Staubli VAL3: francais.pjx

--- francais.pjx ---
Parameters version=s7.1 stackSize=5000 millimeterUnit=true
Program file=message.pgx
Program file=page.pgx
Data file=francais.dtx

--- message.pgx ---
public program message(string& message[], num index)
// English IF message
begin
  // lenght of message
  //
  switch index
    case 0
      message="Voulez-vous entrer dans le:"
    break
    case 1
      message="< SI ASSISTANT >"
    break
    case 2
      message="Sélect. le type de condition pour vérifier"
    break
    case 3
      message="Sélect. l'Entrée"
    break
    case 4
      message="Sélect. la Sortie"
    break
    case 5
      message="Sélect. L'entrée EMAP"
    break
    case 6
      message="Sélect. la voie comment faire fonctionner l'instruction"
    break
    case 7
      message="Sélect. l'instruction pour associer vers le:"
    break
    case 8
      message="Sélect. de la liste le: "
    break
  endSwitch
end

--- page.pgx ---
public program page(string& menuname[], num index)
// set all the page in english IF
begin
  //
  //  PAGE
  //
  switch index
    //
  endSwitch
end
